// TIA Portal V17 export
// export: Created 2023-08-28T22:41:32.6164324Z, ExportSetting WithDefaults, DisplayName Totally Integrated Automation Portal, DisplayVersion V17 Update 5, DisplayName TIA Portal Openness, DisplayVersion V17 Update 5, DisplayName TIA Portal Teamcenter Gateway, DisplayVersion V17 Update 5, DisplayName TIA Portal Version Control Interface, DisplayVersion V17, DisplayName Simotion SCOUT TIA, DisplayVersion 5.4.3.0, DisplayName TIA Portal Test Suite Advanced, DisplayVersion V17 Update 1, DisplayName SIMOCODE ES, DisplayVersion V17 Update 5, DisplayName SINAMICS Startdrive Advanced, DisplayVersion V17 SP1, DisplayName SINAMICS Startdrive G130, G150, S120, S150, SINAMICS MV, S210, DisplayVersion V17 SP1, DisplayName SINAMICS Startdrive G110M, G120, G120C, G120D, G120P, G115D, DisplayVersion V17 SP1, DisplayName SIRIUS Safety ES, DisplayVersion V17 Update 5, DisplayName STEP 7 Professional, DisplayVersion V17 Update 5, DisplayName STEP 7 CFC, DisplayVersion V17 Update 1, DisplayName STEP 7 Safety, DisplayVersion V17, DisplayName WinCC Advanced, DisplayVersion V17 Update 5, DisplayName SIMATIC Visualization Architect, DisplayVersion V17 Update 5
DATA_BLOCK "S1_ESTOP1_DB"   // DB1800, F_DB
// stored: AutoNumber true, DBAccessibleFromOPCUA true, DBAccessibleFromWebserver true, InstanceOfName F_ESTOP1, InstanceOfType FB
"F_ESTOP1 "
BEGIN
END_DATA_BLOCK

DATA_BLOCK "S2_ESTOP1_DB"   // DB1801, F_DB
// stored: AutoNumber true, DBAccessibleFromOPCUA true, DBAccessibleFromWebserver true, InstanceOfName F_ESTOP1, InstanceOfType FB
"F_ESTOP1 "
BEGIN
END_DATA_BLOCK

DATA_BLOCK "S3_ESTOP1_DB"   // DB1802, F_DB
// stored: AutoNumber true, DBAccessibleFromOPCUA true, DBAccessibleFromWebserver true, InstanceOfName F_ESTOP1, InstanceOfType FB
"F_ESTOP1 "
BEGIN
END_DATA_BLOCK

DATA_BLOCK "S4_ESTOP1_DB"   // DB1803, F_DB
// stored: AutoNumber true, DBAccessibleFromOPCUA true, DBAccessibleFromWebserver true, InstanceOfName F_ESTOP1, InstanceOfType FB
"F_ESTOP1 "
BEGIN
END_DATA_BLOCK

DATA_BLOCK "A1_ESTOP1_DB"   // DB1804, F_DB
// stored: AutoNumber true, DBAccessibleFromOPCUA true, DBAccessibleFromWebserver true, InstanceOfName F_ESTOP1, InstanceOfType FB
"F_ESTOP1 "
BEGIN
END_DATA_BLOCK

DATA_BLOCK "A2_ESTOP1_DB"   // DB1805, F_DB
// stored: AutoNumber true, DBAccessibleFromOPCUA true, DBAccessibleFromWebserver true, InstanceOfName F_ESTOP1, InstanceOfType FB
"F_ESTOP1 "
BEGIN
END_DATA_BLOCK

DATA_BLOCK "A3_ESTOP1_DB"   // DB1806, F_DB
// stored: AutoNumber true, DBAccessibleFromOPCUA true, DBAccessibleFromWebserver true, InstanceOfName F_ESTOP1, InstanceOfType FB
"F_ESTOP1 "
BEGIN
END_DATA_BLOCK

DATA_BLOCK "A4_ESTOP1_DB"   // DB1807, F_DB
// stored: AutoNumber true, DBAccessibleFromOPCUA true, DBAccessibleFromWebserver true, InstanceOfName F_ESTOP1, InstanceOfType FB
"F_ESTOP1 "
BEGIN
END_DATA_BLOCK

DATA_BLOCK "A5_ESTOP1_DB"   // DB1808, F_DB
// stored: AutoNumber true, DBAccessibleFromOPCUA true, DBAccessibleFromWebserver true, InstanceOfName F_ESTOP1, InstanceOfType FB
"F_ESTOP1 "
BEGIN
END_DATA_BLOCK

DATA_BLOCK "A6_ESTOP1_DB"   // DB1809, F_DB
// stored: AutoNumber true, DBAccessibleFromOPCUA true, DBAccessibleFromWebserver true, InstanceOfName F_ESTOP1, InstanceOfType FB
"F_ESTOP1 "
BEGIN
END_DATA_BLOCK

DATA_BLOCK "A7_ESTOP1_DB"   // DB1810, F_DB
// stored: AutoNumber true, DBAccessibleFromOPCUA true, DBAccessibleFromWebserver true, InstanceOfName F_ESTOP1, InstanceOfType FB
"F_ESTOP1 "
BEGIN
END_DATA_BLOCK

DATA_BLOCK "L1_ESTOP1_DB"   // DB1811, F_DB
// stored: AutoNumber true, DBAccessibleFromOPCUA true, DBAccessibleFromWebserver true, InstanceOfName F_ESTOP1, InstanceOfType FB
"F_ESTOP1 "
BEGIN
END_DATA_BLOCK

DATA_BLOCK "L2_ESTOP1_DB"   // DB1812, F_DB
// stored: AutoNumber true, DBAccessibleFromOPCUA true, DBAccessibleFromWebserver true, InstanceOfName F_ESTOP1, InstanceOfType FB
"F_ESTOP1 "
BEGIN
END_DATA_BLOCK

DATA_BLOCK "L3_ESTOP1_DB"   // DB1813, F_DB
// stored: AutoNumber true, DBAccessibleFromOPCUA true, DBAccessibleFromWebserver true, InstanceOfName F_ESTOP1, InstanceOfType FB
"F_ESTOP1 "
BEGIN
END_DATA_BLOCK

DATA_BLOCK "L4_ESTOP1_DB"   // DB1814, F_DB
// stored: AutoNumber true, DBAccessibleFromOPCUA true, DBAccessibleFromWebserver true, InstanceOfName F_ESTOP1, InstanceOfType FB
"F_ESTOP1 "
BEGIN
END_DATA_BLOCK

DATA_BLOCK "L5_ESTOP1_DB"   // DB1815, F_DB
// stored: AutoNumber true, DBAccessibleFromOPCUA true, DBAccessibleFromWebserver true, InstanceOfName F_ESTOP1, InstanceOfType FB
"F_ESTOP1 "
BEGIN
END_DATA_BLOCK

DATA_BLOCK "L6_ESTOP1_DB"   // DB1816, F_DB
// stored: AutoNumber true, DBAccessibleFromOPCUA true, DBAccessibleFromWebserver true, InstanceOfName F_ESTOP1, InstanceOfType FB
"F_ESTOP1 "
BEGIN
END_DATA_BLOCK

DATA_BLOCK "L7_ESTOP1_DB"   // DB1817, F_DB
// stored: AutoNumber true, DBAccessibleFromOPCUA true, DBAccessibleFromWebserver true, InstanceOfName F_ESTOP1, InstanceOfType FB
"F_ESTOP1 "
BEGIN
END_DATA_BLOCK

DATA_BLOCK "L8_ESTOP1_DB"   // DB1818, F_DB
// stored: AutoNumber true, DBAccessibleFromOPCUA true, DBAccessibleFromWebserver true, InstanceOfName F_ESTOP1, InstanceOfType FB
"F_ESTOP1 "
BEGIN
END_DATA_BLOCK

DATA_BLOCK "L9_ESTOP1_DB"   // DB1819, F_DB
// stored: AutoNumber true, DBAccessibleFromOPCUA true, DBAccessibleFromWebserver true, InstanceOfName F_ESTOP1, InstanceOfType FB
"F_ESTOP1 "
BEGIN
END_DATA_BLOCK

DATA_BLOCK "L10_ESTOP1_DB"   // DB1820, F_DB
// stored: AutoNumber true, DBAccessibleFromOPCUA true, DBAccessibleFromWebserver true, InstanceOfName F_ESTOP1, InstanceOfType FB
"F_ESTOP1 "
BEGIN
END_DATA_BLOCK

DATA_BLOCK "L11_ESTOP1_DB"   // DB1821, F_DB
// stored: AutoNumber true, DBAccessibleFromOPCUA true, DBAccessibleFromWebserver true, InstanceOfName F_ESTOP1, InstanceOfType FB
"F_ESTOP1 "
BEGIN
END_DATA_BLOCK

DATA_BLOCK "L12_ESTOP1_DB"   // DB1822, F_DB
// stored: AutoNumber true, DBAccessibleFromOPCUA true, DBAccessibleFromWebserver true, InstanceOfName F_ESTOP1, InstanceOfType FB
"F_ESTOP1 "
BEGIN
END_DATA_BLOCK

DATA_BLOCK "L13_ESTOP1_DB"   // DB1823, F_DB
// stored: AutoNumber true, DBAccessibleFromOPCUA true, DBAccessibleFromWebserver true, InstanceOfName F_ESTOP1, InstanceOfType FB
"F_ESTOP1 "
BEGIN
END_DATA_BLOCK

DATA_BLOCK "L14_ESTOP1_DB"   // DB1824, F_DB
// stored: AutoNumber true, DBAccessibleFromOPCUA true, DBAccessibleFromWebserver true, InstanceOfName F_ESTOP1, InstanceOfType FB
"F_ESTOP1 "
BEGIN
END_DATA_BLOCK

DATA_BLOCK "L15_ESTOP1_DB"   // DB1825, F_DB
// stored: AutoNumber true, DBAccessibleFromOPCUA true, DBAccessibleFromWebserver true, InstanceOfName F_ESTOP1, InstanceOfType FB
"F_ESTOP1 "
BEGIN
END_DATA_BLOCK
